(* IEC 61131-3 sources: SafePLC-Gen-Evaluation/PatchEvaluation-DEXPI-XML, 2 files *)

(* ---- io_declarations.st ---- *)
(* ==================================================  *)
(* PLC I/O Variable Declarations — CODESYS 3.5  *)
(* Generated by SafePLC-Gen Multimodal  *)
(* ==================================================  *)

VAR_GLOBAL
    (* --- Analog Inputs ---  *)
    PI_4712.01_Raw               AT %IW0       : INT := 0;    (* PI-4712.01 — PI-4712.01 — Field  *)
    PICSA_4712.02_Raw            AT %IW2       : INT := 0;    (* PICSA-4712.02 — PICSA-4712.02 — CentralLocation  *)
    TICSA_4750.03_Raw            AT %IW4       : INT := 0;    (* TICSA-4750.03 — TICSA-4750.03 — CentralLocation  *)
    (* --- Analog Outputs ---  *)
    PV4712.02_Out                AT %QW0       : INT := 0;    (* PV4712.02 — PV4712.02  *)
    TV4750.03_Out                AT %QW2       : INT := 0;    (* TV4750.03 — TV4750.03  *)
    (* --- Digital Inputs ---  *)
    HS_4750.01                   AT %IX0.0     : BOOL := FALSE;    (* HS-4750.01 — HS-4750.01 — CentralLocation  *)
END_VAR

(* ---- generated_code.st ---- *)
(* Generated by SafePLC-Gen Multimodal — CODESYS 3.5 *)
(* IEC 61131-3 Structured Text *)
(* Date: 2026-04-15T12:28:46.434167 *)

PROGRAM Control_System

VAR
    (* AT-addressed I/O variables *)
    PI_4712_01_Raw               AT %IW0       : INT := 0;
    PICSA_4712_02_Raw            AT %IW2       : INT := 0;
    TICSA_4750_03_Raw            AT %IW4       : INT := 0;
    PV4712_02_Out                AT %QW0       : INT := 0;
    TV4750_03_Out                AT %QW2       : INT := 0;
    HS_4750_01                   AT %IX0.0     : BOOL := FALSE;
END_VAR

VAR
    (* Internal variables *)
    FirstScan                    : BOOL := TRUE;

    (* Scaled process variables *)
    PI_4712_01_Scaled            : REAL := 0.0;
    PICSA_4712_02_Scaled         : REAL := 0.0;
    TICSA_4750_03_Scaled         : REAL := 0.0;

    (* Alarm setpoints *)
    PI_4712_01_HH_SP             : REAL := 150.0;
    PI_4712_01_H_SP              : REAL := 120.0;
    PI_4712_01_L_SP              : REAL := 20.0;
    PI_4712_01_LL_SP             : REAL := 10.0;
    PI_4712_01_Deadband          : REAL := 2.0;

    PICSA_4712_02_HH_SP          : REAL := 150.0;
    PICSA_4712_02_H_SP           : REAL := 120.0;
    PICSA_4712_02_L_SP           : REAL := 20.0;
    PICSA_4712_02_LL_SP          : REAL := 10.0;
    PICSA_4712_02_Deadband       : REAL := 2.0;

    TICSA_4750_03_HH_SP          : REAL := 80.0;
    TICSA_4750_03_H_SP           : REAL := 70.0;
    TICSA_4750_03_L_SP           : REAL := 30.0;
    TICSA_4750_03_LL_SP          : REAL := 20.0;
    TICSA_4750_03_Deadband       : REAL := 1.0;

    (* Alarm states *)
    PI_4712_01_HH_Latch          : SR := (S1 := FALSE, R := FALSE);
    PI_4712_01_LL_Latch          : SR := (S1 := FALSE, R := FALSE);
    PI_4712_01_H                 : BOOL := FALSE;
    PI_4712_01_L                 : BOOL := FALSE;

    PICSA_4712_02_HH_Latch       : SR := (S1 := FALSE, R := FALSE);
    PICSA_4712_02_LL_Latch       : SR := (S1 := FALSE, R := FALSE);
    PICSA_4712_02_H              : BOOL := FALSE;
    PICSA_4712_02_L              : BOOL := FALSE;

    TICSA_4750_03_HH_Latch       : SR := (S1 := FALSE, R := FALSE);
    TICSA_4750_03_LL_Latch       : SR := (S1 := FALSE, R := FALSE);
    TICSA_4750_03_H              : BOOL := FALSE;
    TICSA_4750_03_L              : BOOL := FALSE;

    (* Control loop variables *)
    PICSA_4712_02_SP             : REAL := 100.0;
    PICSA_4712_02_Error          : REAL := 0.0;
    PICSA_4712_02_Kp             : REAL := 2.0;
    PICSA_4712_02_Ki             : REAL := 0.1;
    PICSA_4712_02_Integral       : REAL := 0.0;
    PICSA_4712_02_Output         : REAL := 0.0;

    TICSA_4750_03_SP             : REAL := 60.0;
    TICSA_4750_03_Error          : REAL := 0.0;
    TICSA_4750_03_Kp             : REAL := 1.5;
    TICSA_4750_03_Ki             : REAL := 0.05;
    TICSA_4750_03_Integral       : REAL := 0.0;
    TICSA_4750_03_Output         : REAL := 0.0;

    (* Acknowledgement inputs *)
    PI_4712_01_HH_Ack            : BOOL := FALSE;
    PI_4712_01_LL_Ack            : BOOL := FALSE;
    PICSA_4712_02_HH_Ack         : BOOL := FALSE;
    PICSA_4712_02_LL_Ack         : BOOL := FALSE;
    TICSA_4750_03_HH_Ack         : BOOL := FALSE;
    TICSA_4750_03_LL_Ack         : BOOL := FALSE;

    (* System alarm aggregation *)
    System_Alarm                 : BOOL := FALSE;
END_VAR

(* First-scan initialization *)
IF FirstScan THEN
    PV4712_02_Out := 6554;
    TV4750_03_Out := 6554;
    PICSA_4712_02_Integral := 0.0;
    TICSA_4750_03_Integral := 0.0;
    FirstScan := FALSE;
    RETURN;
END_IF;

(* Scale analog inputs from 4-20 mA to engineering units *)
PI_4712_01_Scaled := ((INT_TO_REAL(PI_4712_01_Raw) - 6554.0) / (32767.0 - 6554.0)) * 200.0 + 0.0;
PICSA_4712_02_Scaled := ((INT_TO_REAL(PICSA_4712_02_Raw) - 6554.0) / (32767.0 - 6554.0)) * 200.0 + 0.0;
TICSA_4750_03_Scaled := ((INT_TO_REAL(TICSA_4750_03_Raw) - 6554.0) / (32767.0 - 6554.0)) * 100.0 + 0.0;

(* PI-4712.01 Four-level alarm logic with deadband *)
IF PI_4712_01_Scaled >= PI_4712_01_HH_SP THEN
    PI_4712_01_HH_Latch.S1 := TRUE;
ELSIF PI_4712_01_Scaled <= (PI_4712_01_HH_SP - PI_4712_01_Deadband) THEN
    PI_4712_01_HH_Latch.S1 := FALSE;
END_IF;

IF PI_4712_01_HH_Ack AND (PI_4712_01_Scaled <= (PI_4712_01_HH_SP - PI_4712_01_Deadband)) THEN
    PI_4712_01_HH_Latch.R := TRUE;
END_IF;
PI_4712_01_HH_Latch();
PI_4712_01_HH_Latch.R := FALSE;

IF PI_4712_01_Scaled <= PI_4712_01_LL_SP THEN
    PI_4712_01_LL_Latch.S1 := TRUE;
ELSIF PI_4712_01_Scaled >= (PI_4712_01_LL_SP + PI_4712_01_Deadband) THEN
    PI_4712_01_LL_Latch.S1 := FALSE;
END_IF;

IF PI_4712_01_LL_Ack AND (PI_4712_01_Scaled >= (PI_4712_01_LL_SP + PI_4712_01_Deadband)) THEN
    PI_4712_01_LL_Latch.R := TRUE;
END_IF;
PI_4712_01_LL_Latch();
PI_4712_01_LL_Latch.R := FALSE;

IF PI_4712_01_Scaled >= PI_4712_01_H_SP THEN
    PI_4712_01_H := TRUE;
ELSIF PI_4712_01_Scaled <= (PI_4712_01_H_SP - PI_4712_01_Deadband) THEN
    PI_4712_01_H := FALSE;
END_IF;

IF PI_4712_01_Scaled <= PI_4712_01_L_SP THEN
    PI_4712_01_L := TRUE;
ELSIF PI_4712_01_Scaled >= (PI_4712_01_L_SP + PI_4712_01_Deadband) THEN
    PI_4712_01_L := FALSE;
END_IF;

(* PICSA-4712.02 Four-level alarm logic with deadband *)
IF PICSA_4712_02_Scaled >= PICSA_4712_02_HH_SP THEN
    PICSA_4712_02_HH_Latch.S1 := TRUE;
ELSIF PICSA_4712_02_Scaled <= (PICSA_4712_02_HH_SP - PICSA_4712_02_Deadband) THEN
    PICSA_4712_02_HH_Latch.S1 := FALSE;
END_IF;

IF PICSA_4712_02_HH_Ack AND (PICSA_4712_02_Scaled <= (PICSA_4712_02_HH_SP - PICSA_4712_02_Deadband)) THEN
    PICSA_4712_02_HH_Latch.R := TRUE;
END_IF;
PICSA_4712_02_HH_Latch();
PICSA_4712_02_HH_Latch.R := FALSE;

IF PICSA_4712_02_Scaled <= PICSA_4712_02_LL_SP THEN
    PICSA_4712_02_LL_Latch.S1 := TRUE;
ELSIF PICSA_4712_02_Scaled >= (PICSA_4712_02_LL_SP + PICSA_4712_02_Deadband) THEN
    PICSA_4712_02_LL_Latch.S1 := FALSE;
END_IF;

IF PICSA_4712_02_LL_Ack AND (PICSA_4712_02_Scaled >= (PICSA_4712_02_LL_SP + PICSA_4712_02_Deadband)) THEN
    PICSA_4712_02_LL_Latch.R := TRUE;
END_IF;
PICSA_4712_02_LL_Latch();
PICSA_4712_02_LL_Latch.R := FALSE;

IF PICSA_4712_02_Scaled >= PICSA_4712_02_H_SP THEN
    PICSA_4712_02_H := TRUE;
ELSIF PICSA_4712_02_Scaled <= (PICSA_4712_02_H_SP - PICSA_4712_02_Deadband) THEN
    PICSA_4712_02_H := FALSE;
END_IF;

IF PICSA_4712_02_Scaled <= PICSA_4712_02_L_SP THEN
    PICSA_4712_02_L := TRUE;
ELSIF PICSA_4712_02_Scaled >= (PICSA_4712_02_L_SP + PICSA_4712_02_Deadband) THEN
    PICSA_4712_02_L := FALSE;
END_IF;

(* TICSA-4750.03 Four-level alarm logic with deadband *)
IF TICSA_4750_03_Scaled >= TICSA_4750_03_HH_SP THEN
    TICSA_4750_03_HH_Latch.S1 := TRUE;
ELSIF TICSA_4750_03_Scaled <= (TICSA_4750_03_HH_SP - TICSA_4750_03_Deadband) THEN
    TICSA_4750_03_HH_Latch.S1 := FALSE;
END_IF;

IF TICSA_4750_03_HH_Ack AND (TICSA_4750_03_Scaled <= (TICSA_4750_03_HH_SP - TICSA_4750_03_Deadband)) THEN
    TICSA_4750_03_HH_Latch.R := TRUE;
END_IF;
TICSA_4750_03_HH_Latch();
TICSA_4750_03_HH_Latch.R := FALSE;

IF TICSA_4750_03_Scaled <= TICSA_4750_03_LL_SP THEN
    TICSA_4750_03_LL_Latch.S1 := TRUE;
ELSIF TICSA_4750_03_Scaled >= (TICSA_4750_03_LL_SP + TICSA_4750_03_Deadband) THEN
    TICSA_4750_03_LL_Latch.S1 := FALSE;
END_IF;

IF TICSA_4750_03_LL_Ack AND (TICSA_4750_03_Scaled >= (TICSA_4750_03_LL_SP + TICSA_4750_03_Deadband)) THEN
    TICSA_4750_03_LL_Latch.R := TRUE;
END_IF;
TICSA_4750_03_LL_Latch();
TICSA_4750_03_LL_Latch.R := FALSE;

IF TICSA_4750_03_Scaled >= TICSA_4750_03_H_SP THEN
    TICSA_4750_03_H := TRUE;
ELSIF TICSA_4750_03_Scaled <= (TICSA_4750_03_H_SP - TICSA_4750_03_Deadband) THEN
    TICSA_4750_03_H := FALSE;
END_IF;

IF TICSA_4750_03_Scaled <= TICSA_4750_03_L_SP THEN
    TICSA_4750_03_L := TRUE;
ELSIF TICSA_4750_03_Scaled >= (TICSA_4750_03_L_SP + TICSA_4750_03_Deadband) THEN
    TICSA_4750_03_L := FALSE;
END_IF;

(* PICSA-4712.02 Pressure control loop - PI controller *)
PICSA_4712_02_Error := PICSA_4712_02_SP - PICSA_4712_02_Scaled;

PICSA_4712_02_Integral := PICSA_4712_02_Integral + (PICSA_4712_02_Ki * PICSA_4712_02_Error);
IF PICSA_4712_02_Integral > 100.0 THEN
    PICSA_4712_02_Integral := 100.0;
ELSIF PICSA_4712_02_Integral < 0.0 THEN
    PICSA_4712_02_Integral := 0.0;
END_IF;

PICSA_4712_02_Output := (PICSA_4712_02_Kp * PICSA_4712_02_Error) + PICSA_4712_02_Integral;

IF PICSA_4712_02_Output > 100.0 THEN
    PICSA_4712_02_Output := 100.0;
ELSIF PICSA_4712_02_Output < 0.0 THEN
    PICSA_4712_02_Output := 0.0;
END_IF;

PV4712_02_Out := REAL_TO_INT(6554.0 + (PICSA_4712_02_Output / 100.0) * (32767.0 - 6554.0));

(* TICSA-4750.03 Temperature control loop - PI controller *)
IF HS_4750_01 THEN
    TICSA_4750_03_Error := TICSA_4750_03_SP - TICSA_4750_03_Scaled;

    TICSA_4750_03_Integral := TICSA_4750_03_Integral + (TICSA_4750_03_Ki * TICSA_4750_03_Error);
    IF TICSA_4750_03_Integral > 100.0 THEN
        TICSA_4750_03_Integral := 100.0;
    ELSIF TICSA_4750_03_Integral < 0.0 THEN
        TICSA_4750_03_Integral := 0.0;
    END_IF;

    TICSA_4750_03_Output := (TICSA_4750_03_Kp * TICSA_4750_03_Error) + TICSA_4750_03_Integral;

    IF TICSA_4750_03_Output > 100.0 THEN
        TICSA_4750_03_Output := 100.0;
    ELSIF TICSA_4750_03_Output < 0.0 THEN
        TICSA_4750_03_Output := 0.0;
    END_IF;

    TV4750_03_Out := REAL_TO_INT(6554.0 + (TICSA_4750_03_Output / 100.0) * (32767.0 - 6554.0));
ELSE
    TV4750_03_Out := 6554;
    TICSA_4750_03_Integral := 0.0;
END_IF;

(* Aggregate all alarm states *)
System_Alarm :=
    PI_4712_01_HH_Latch.Q1 OR PI_4712_01_LL_Latch.Q1 OR
    PI_4712_01_H OR PI_4712_01_L OR
    PICSA_4712_02_HH_Latch.Q1 OR PICSA_4712_02_LL_Latch.Q1 OR
    PICSA_4712_02_H OR PICSA_4712_02_L OR
    TICSA_4750_03_HH_Latch.Q1 OR TICSA_4750_03_LL_Latch.Q1 OR
    TICSA_4750_03_H OR TICSA_4750_03_L;

END_PROGRAM
